Omron Sysmac Studio project Encoder (Sysmac Studio 1.23.0.14, StandardProject)

# Controller new_Controller_0: NX1P2-1040DT1 version 1.18
Task PrimaryTask (priority 4, period or condition 2000): Programa0

VAR_GLOBAL
    PP : BOOL;  (* at BuiltInIO://cpu/#0/Input_Bit_00 *)
    PM : BOOL;  (* at BuiltInIO://cpu/#0/Input_Bit_01 *)
    PR : BOOL;  (* at BuiltInIO://cpu/#0/Input_Bit_02 *)
    CounterEnable : BOOL;  (* at IOBus://unit#1/Ch1 Encoder Counter Operation Command/Ch1 Counter Enable *)
    ZEnable : BOOL;  (* at IOBus://unit#1/Ch1 Encoder Counter Operation Command/Ch1 Phase Z Reset Enable *)
    ExtEnable : BOOL;
    CounterReset : BOOL;  (* at IOBus://unit#1/Ch1 Encoder Counter Operation Command/Ch1 Internal Reset Execution *)
    CounterPreset : BOOL;  (* at IOBus://unit#1/Ch1 Encoder Counter Operation Command/Ch1 Preset Execution *)
    ZCompleted : BOOL;  (* at IOBus://unit#1/Ch1 Reset/External Input Status/Ch1 Phase Z Reset Completed Flag *)
    Preset : DINT;  (* at IOBus://unit#1/Ch1 Preset Command Value *)
END_VAR

PROGRAM Programa0
VAR_EXTERNAL
    PM : BOOL;
    CounterEnable : BOOL;
    PP : BOOL;
    ZEnable : BOOL;
    ExtEnable : BOOL;
    PR : BOOL;
    CounterReset : BOOL;
    CounterPreset : BOOL;
    ZCompleted : BOOL;
    Preset : DINT;
END_VAR

(* Section Sección0: ladder, written here as Structured Text *)

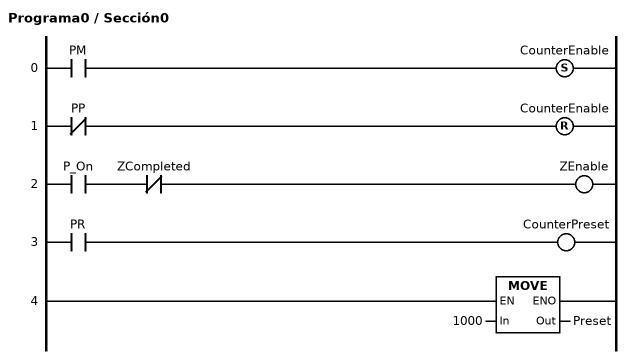
(* Rung 0 *)
IF PM THEN CounterEnable := TRUE; END_IF;
(* Rung 1 *)
IF NOT PP THEN CounterEnable := FALSE; END_IF;
(* Rung 2 *)
ZEnable := P_On AND NOT ZCompleted;
(* Rung 3 *)
CounterPreset := PR;
(* Rung 4 *)
Preset := 1000;
END_PROGRAM